(*

.. <legal notes>

legal notes
=================
| SPDX-FileCopyrightText: © 2026 Oleksandr Tiutyk <trofimich@gmail.com>
| SPDX-License-Identifier: LGPL-3.0-only
| For details check: LGPL-3.0-only_

.. _LGPL-3.0-only: https://www.gnu.org/licenses/lgpl-3.0.en.html

.. </legal notes>

*)

FUNCTION_BLOCK ABSTRACT Device EXTENDS AutomationComponent IMPLEMENTS IChildAutomationComponent

METHOD FB_init : BOOL
VAR_INPUT
	(* if TRUE, the retain variables are initialized (warm start / cold start)*)
	bInitRetains	: BOOL;
	(* if TRUE, the instance afterwards gets moved into the copy code (online change)*)
	bInCopyCode	: BOOL;
	name : WSTRING;
	parent : IParentAutomationComponent;
END_VAR
_Parent := parent;
END_METHOD

{attribute 'monitoring' := 'call'}
PROPERTY FINAL Parent : IParentAutomationComponent
GET
Parent := _Parent;
END_GET
END_PROPERTY

END_FUNCTION_BLOCK

(* stored: Version 1.1.0.1
   POU Device: Id {f3b4f1f5-d7e8-495b-a404-a87157d5f32f}, SpecialFunc None
   Method FB_init: Id {6e7d33a1-6d80-43ad-a8d8-899454af5a81}
   Property Parent: Id {9a2a0d18-500c-4856-b3bd-133e8d7de4d2}
   Get Get: Id {5e19e287-9498-42dd-bbfe-2069a9e5105e} *)
